TYPE MotorType :
(
	MotorType_Default	 	:= 0, 		//增量式编码器(需要执行McHome)
	MotorType_DDmotor_HC 	:= 1,		//横川DD马达(不需要执行McHome,使用高创驱动器自带的回原点方式)
	MotorType_Absolute		:= 2		//绝对式编码器(不需要执行McHome)
)UINT;
END_TYPE

(* stored: Version 1.1.0.1, ProductVersion 3.1.4024.4
   DUT MotorType: Id {45234b17-1d1e-4e33-a150-3db7dd4769cc} *)
